FUNCTION_BLOCK PUT_WORD (* Writes a bit value into a WORD *)
  (* Standard: 61499-1; Classification: Math; Function: Bit put; Type: WORD *)
  (* Version 0.0, 2008-01-20, JHC, Holobloc Inc *)
  (* Compiler header: package fb.rt.math; *)
  (* Compiler Java Sun JDK 1.6.0 *)
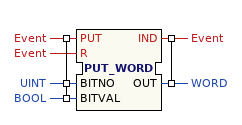
  EVENT_INPUT
    PUT WITH BITVAL, BITNO; (* Write BITVAL to BITNO of OUT *)
    R; (* Reset OUT to 0 *)
  END_EVENT
  EVENT_OUTPUT
    IND WITH OUT; (* OUT value changed or reset *)
  END_EVENT
  VAR_INPUT
    BITNO : UINT; (* Bit number (modulo 16) of OUT to which to write BITVAL *)
    BITVAL : BOOL; (* Bit value to write to OUT *)
  END_VAR
  VAR_OUTPUT
    OUT : WORD; (* The output value *)
  END_VAR
  ALGORITHM PUT IN Java: (* Write BITVAL to BITNO of WORD *)
IND.serviceEvent(this);
  END_ALGORITHM
  ALGORITHM R IN ST: (* Reset OUT to 0 *)
OUT := 0;
IND.serviceEvent(this);
  END_ALGORITHM
END_FUNCTION_BLOCK
